{attribute 'hide_all_locals'}
{attribute 'conditionalshow'}
FUNCTION_BLOCK FB_Generator
VAR_INPUT
	{attribute 'hide'}
	bEnable								: BOOL;									//Enable or disable this function
	{attribute 'hide'}
	bError								: BOOL;									//Generator has a error
	{attribute 'hide'}
	bWarning							: BOOL;									//Generator has a warning
	{attribute 'hide'}
	bReset								: BOOL;									//Reset the function after a error (Read the Reset output back with a negative edge because send a active reset signal to the generator)
	{attribute 'hide'}
	bWriteWithDelay						: BOOL;									//Write with Delay the Data to the output (Not al Output Data is writen with Delay)
	{attribute 'hide'}
	iErrorCode							: INT;									//Error Code from external Generator
	{attribute 'hide'}
	iWarningCode						: INT;									//Warning Code from external Generator
	{attribute 'hide'}
	dwBatterySOC						: DWORD;								//Actual Battery SOC in %
	{attribute 'hide'}
	lrTotalCounterEnergy_Consumption	: LREAL;								//Total Counter for Energy consumption with unit Wh
	{attribute 'hide'}
	lrTotalCounterEnergy_Production		: LREAL;								//Total Counter for Energy production with unit Wh
	{attribute 'hide'}
	lrCounterEnergyT1_Consumption		: LREAL;								//Total counter for energy Tariff 1 consumption with unit Wh
	{attribute 'hide'}
	lrCounterEnergyT2_Consumption		: LREAL;								//Total counter for energy Tariff 2 consumption with unit Wh
	{attribute 'hide'}
	lrCounterEnergyT1_Production		: LREAL;								//Total counter for energy Tariff 1 production with unit Wh
	{attribute 'hide'}
	lrCounterEnergyT2_Production		: LREAL;								//Total counter for energy Tariff 2 production with unit Wh
	{attribute 'hide'}
	lrPowerGenerator					: LREAL;								//Input Value from the power of the Generator with unit W
	{attribute 'hide'}
	tDelaySwitchOn						: TIME;									//Delay befor the generator is switching on
	{attribute 'hide'}
	tTimDelayOutput						: TIME := T#5S;							//Delay Time to write some Data to the Output
	{attribute 'hide'}
	stSetupGenerator					: ST_Setup_Generator;					//Setup Generator
END_VAR
VAR_OUTPUT
	{attribute 'hide'}
	stDataGeneratorOut					: ST_Generator_Output;					//Generator Output data
	{attribute 'hide'}
	stDataGeneratorOutDelay				: ST_Generator_Output;					//Generator Output data with delay
END_VAR
VAR
	FPReset								: R_TRIG;								//Internal positive edge
	FPResetIntern						: R_TRIG;								//Internal positive edge
	FPEnable							: R_TRIG;								//Internal positive Edge
	FNEnable							: F_TRIG;								//Internal negative Edge
	timDelayOutputs						: TON;									//Timer to send Data with Delay to the outputs
	timGenEin							: TON;									//Timer to switch on the generator
	timResetOut							: TOF;									//Timer Reset Out
END_VAR

//Creator : Kai Ebensperger
//Company : Lynus AG
//Date : 28.05.2021
//Version : 1.0.0.0

//With this function its possible to control the basics from a generator
//The generator is switching on and off with the SOC from the battery

(*---------------------------------------------------------------Limit Inputs-------------------------------------------------------------------------------*)

dwBatterySOC := LIMIT(0,dwBatterySOC,100);

IF stSetupGenerator.byEnableSOC > stSetupGenerator.byDisableSOC THEN stSetupGenerator.byDisableSOC := stSetupGenerator.byEnableSOC + 1; END_IF

stSetupGenerator.byDisableSOC := LIMIT(1,stSetupGenerator.byDisableSOC,100);
	stSetupGenerator.byEnableSOC := LIMIT(0,stSetupGenerator.byEnableSOC,100);
		tDelaySwitchOn := LIMIT(T#10S,tDelaySwitchOn,T#2M);
		
IF IsFinite(F_LREAL(lrTotalCounterEnergy_Consumption)) THEN lrTotalCounterEnergy_Consumption := LIMIT(0,lrTotalCounterEnergy_Consumption,999999999999999); END_IF
	IF IsFinite(F_LREAL(lrTotalCounterEnergy_Production)) THEN lrTotalCounterEnergy_Production := LIMIT(0,lrTotalCounterEnergy_Production,999999999999999); END_IF
		IF IsFinite(F_LREAL(lrCounterEnergyT1_Consumption)) THEN lrCounterEnergyT1_Consumption := LIMIT(0,lrCounterEnergyT1_Consumption,999999999999999); END_IF
			IF IsFinite(F_LREAL(lrCounterEnergyT2_Consumption)) THEN lrCounterEnergyT2_Consumption := LIMIT(0,lrCounterEnergyT2_Consumption,999999999999999); END_IF
				IF IsFinite(F_LREAL(lrCounterEnergyT1_Production)) THEN lrCounterEnergyT1_Production := LIMIT(0,lrCounterEnergyT1_Production,999999999999999); END_IF
					IF IsFinite(F_LREAL(lrCounterEnergyT2_Production)) THEN lrCounterEnergyT2_Production := LIMIT(0,lrCounterEnergyT2_Production,999999999999999); END_IF
						lrPowerGenerator := LIMIT(-999999999999999,lrPowerGenerator,999999999999999);
	
(*---------------------------------------------------------------------------enable----------------------------------------------------------------------------------*)

stDataGeneratorOut.bEnabled := bEnable;

(*-----------------------------------------------------------------------------Error-Warning and Reset----------------------------------------------------------------------------*)

IF bWarning THEN stDataGeneratorOut.byErrorWarning := 1; END_IF 
	IF bError THEN stDataGeneratorOut.byErrorWarning := 2; END_IF

FPReset(CLK:= stSetupGenerator.bReset AND stDataGeneratorOut.byErrorWarning <> 0, Q=> ); 

timResetOut(IN:= FPReset.Q, PT:= T#2S, Q=> , ET=> );	

	stDataGeneratorOut.bSReset := timResetOut.Q;

FPResetIntern(CLK:= bReset, Q=> );	
	
IF NOT bError AND NOT bWarning AND FPResetIntern.Q THEN stDataGeneratorOut.byErrorWarning := 0; END_IF

//Messages and Error Codes
IF stDataGeneratorOut.byErrorWarning = 1 AND iWarningCode = 0 THEN stDataGeneratorOut.eMessage := E_Message_Generator.eNoConnectionToBackend;
ELSIF stDataGeneratorOut.byErrorWarning = 2 AND iErrorCode = 0 THEN stDataGeneratorOut.eMessage := E_Message_Generator.eGeneratorError;
ELSIF stDataGeneratorOut.byErrorWarning = 2 AND iErrorCode = 1 THEN stDataGeneratorOut.eMessage := E_Message_Generator.eTooMuchGenerators;
ELSE stDataGeneratorOut.eMessage := E_Message_Generator.eNoMessage; 
END_IF

(*----------------------------------------------------------------------------Logic------------------------------------------------------------------------------------*)

//Switch on
timGenEin(IN:= bEnable AND stDataGeneratorOut.byErrorWarning <> 2 AND dwBatterySOC <= stSetupGenerator.byEnableSOC, PT:= tDelaySwitchOn, Q=> , ET=> );
IF timGenEin.Q THEN stDataGeneratorOut.bOutput := TRUE; END_IF 

//Switch off
IF NOT bEnable OR stDataGeneratorOut.byErrorWarning = 2 OR dwBatterySOC >= stSetupGenerator.byDisableSOC THEN stDataGeneratorOut.bOutput := FALSE; END_IF 

(*------------------------------------------------------------------Power Data----------------------------------------------------------------------------------------------*)

timDelayOutputs(IN:= bWriteWithDelay AND bEnable AND NOT timDelayOutputs.Q, PT:= tTimDelayOutput, Q=> , ET=> );
	FPEnable(CLK:= bEnable, Q=> );
		FNEnable(CLK:= bEnable, Q=> );

IF bEnable THEN
	stDataGeneratorOut.lrPower:= LINT_TO_LREAL(LREAL_TO_LINT((lrPowerGenerator / 1000) * 100)) / 100;
		IF IsFinite(F_LREAL(lrCounterEnergyT1_Consumption)) THEN stDataGeneratorOut.lrCounterEnergyT1_Consumption := LINT_TO_LREAL(LREAL_TO_LINT((lrCounterEnergyT1_Consumption / 1000) * 100)) / 100; END_IF
			IF IsFinite(F_LREAL(lrCounterEnergyT2_Consumption)) THEN stDataGeneratorOut.lrCounterEnergyT2_Consumption := LINT_TO_LREAL(LREAL_TO_LINT((lrCounterEnergyT2_Consumption / 1000) * 100)) / 100; END_IF
				IF IsFinite(F_LREAL(lrCounterEnergyT1_Production)) THEN stDataGeneratorOut.lrCounterEnergyT1_Production := LINT_TO_LREAL(LREAL_TO_LINT((lrCounterEnergyT1_Production / 1000) * 100)) / 100; END_IF
					IF IsFinite(F_LREAL(lrCounterEnergyT2_Production)) THEN stDataGeneratorOut.lrCounterEnergyT2_Production := LINT_TO_LREAL(LREAL_TO_LINT((lrCounterEnergyT2_Production / 1000) * 100)) / 100; END_IF
						IF IsFinite(F_LREAL(lrTotalCounterEnergy_Consumption)) THEN stDataGeneratorOut.lrTotalCounterEnergy_Consumption := LINT_TO_LREAL(LREAL_TO_LINT((lrTotalCounterEnergy_Consumption / 1000) * 100)) / 100; END_IF
							IF IsFinite(F_LREAL(lrTotalCounterEnergy_Production)) THEN stDataGeneratorOut.lrTotalCounterEnergy_Production := LINT_TO_LREAL(LREAL_TO_LINT((lrTotalCounterEnergy_Production / 1000) * 100)) / 100; END_IF 	
			
	IF stDataGeneratorOut.lrPower < 0 THEN
		stDataGeneratorOut.lrPowerProduction := 0;
		stDataGeneratorOut.lrPowerConsumption := (stDataGeneratorOut.lrPower * - 1);
	ELSIF stDataGeneratorOut.lrPower > 0 THEN
		stDataGeneratorOut.lrPowerProduction := stDataGeneratorOut.lrPower;
		stDataGeneratorOut.lrPowerConsumption := 0;
	ELSIF stDataGeneratorOut.lrPower = 0 THEN
		stDataGeneratorOut.lrPowerProduction := 0;
		stDataGeneratorOut.lrPowerConsumption := 0;
	END_IF
ELSE	
	stDataGeneratorOut.lrPower := 0;
		stDataGeneratorOut.lrCounterEnergyT1_Consumption := 0;
			stDataGeneratorOut.lrCounterEnergyT2_Consumption := 0;
				stDataGeneratorOut.lrCounterEnergyT1_Production := 0;
					stDataGeneratorOut.lrCounterEnergyT2_Production := 0;
						stDataGeneratorOut.lrPowerProduction := 0;
							stDataGeneratorOut.lrPowerConsumption := 0;	
								stDataGeneratorOut.lrTotalCounterEnergy_Consumption := 0;
									stDataGeneratorOut.lrTotalCounterEnergy_Production := 0;
END_IF

(*---------------------------------------------------------------Outputs-------------------------------------------------------------------------------*)

//Write with Delay or without
IF (bWriteWithDelay AND (timDelayOutputs.Q OR FPEnable.Q OR FNEnable.Q)) OR NOT bWriteWithDelay THEN
	stDataGeneratorOutDelay := stDataGeneratorOut; 
END_IF

END_FUNCTION_BLOCK

(* stored: Version 1.1.0.1, ProductVersion 3.1.4024.9
   POU FB_Generator: Id {ae2fbe09-bbce-45e7-a981-a56d9c79a1e6}, SpecialFunc None *)
